// TIA Portal V18 export
// export: Created 2026-06-08T03:54:34.4007583Z, ExportSetting WithDefaults, DisplayName Totally Integrated Automation Portal, DisplayVersion V18, DisplayName TIA Portal Openness, DisplayVersion V18, DisplayName TIA Portal Version Control Interface, DisplayVersion V18, DisplayName STEP 7 Professional, DisplayVersion V18, DisplayName STEP 7 Safety, DisplayVersion V18, DisplayName WinCC Professional, DisplayVersion V18
VAR_GLOBAL   // PLC tag table "PLC_Tags"
   FT3210_Bon3 AT %ID128 : Real;   // Cảm biến lưu lượng nước dosing vào Bồn 3
   FT3210_Bon3_HMI AT %MD756 : Real;   // Giá trị mô phỏng/HMI song song cho Cảm biến lưu lượng nước dosing vào Bồn 3
   FT3210_Bon3_Use_HMI AT %M420.7 : Bool;   // Chọn chế độ mô phỏng HMI cho Cảm biến lưu lượng nước dosing vào Bồn 3
   FT3210_Bon3_Sim_Req AT %M323.0 : Bool;   // Yêu cầu mô phỏng cảm biến cho Cảm biến lưu lượng nước dosing vào Bồn 3
   FT3210_Bon3_Sim_Active AT %M323.1 : Bool;   // Mô phỏng cảm biến đang hoạt động cho Cảm biến lưu lượng nước dosing vào Bồn 3
   FT3210_Bon3_Eff AT %MD760 : Real;   // Giá trị thực tế/mô phỏng hiệu dụng cho Cảm biến lưu lượng nước dosing vào Bồn 3
   LT3213_Bon3 AT %ID132 : Real;   // Cảm biến mức liên tục Bồn 3
   LT3213_Bon3_HMI AT %MD764 : Real;   // Giá trị mô phỏng/HMI song song cho Cảm biến mức liên tục Bồn 3
   LT3213_Bon3_Use_HMI AT %M421.0 : Bool;   // Chọn chế độ mô phỏng HMI cho Cảm biến mức liên tục Bồn 3
   LT3213_Bon3_Sim_Req AT %M323.2 : Bool;   // Yêu cầu mô phỏng cảm biến cho Cảm biến mức liên tục Bồn 3
   LT3213_Bon3_Sim_Active AT %M323.3 : Bool;   // Mô phỏng cảm biến đang hoạt động cho Cảm biến mức liên tục Bồn 3
   LT3213_Bon3_Eff AT %MD768 : Real;   // Giá trị thực tế/mô phỏng hiệu dụng cho Cảm biến mức liên tục Bồn 3
   TT3214_Bon3 AT %ID136 : Real;   // Cảm biến nhiệt độ Bồn 3
   TT3214_Bon3_HMI AT %MD772 : Real;   // Giá trị mô phỏng/HMI song song cho Cảm biến nhiệt độ Bồn 3
   TT3214_Bon3_Use_HMI AT %M421.1 : Bool;   // Chọn chế độ mô phỏng HMI cho Cảm biến nhiệt độ Bồn 3
   TT3214_Bon3_Sim_Req AT %M323.4 : Bool;   // Yêu cầu mô phỏng cảm biến cho Cảm biến nhiệt độ Bồn 3
   TT3214_Bon3_Sim_Active AT %M323.5 : Bool;   // Mô phỏng cảm biến đang hoạt động cho Cảm biến nhiệt độ Bồn 3
   TT3214_Bon3_Eff AT %MD776 : Real;   // Giá trị thực tế/mô phỏng hiệu dụng cho Cảm biến nhiệt độ Bồn 3
   FT3215_Bon4 AT %ID140 : Real;   // Cảm biến lưu lượng nước dosing vào Bồn 4
   FT3215_Bon4_HMI AT %MD780 : Real;   // Giá trị mô phỏng/HMI song song cho Cảm biến lưu lượng nước dosing vào Bồn 4
   FT3215_Bon4_Use_HMI AT %M421.2 : Bool;   // Chọn chế độ mô phỏng HMI cho Cảm biến lưu lượng nước dosing vào Bồn 4
   FT3215_Bon4_Sim_Req AT %M323.6 : Bool;   // Yêu cầu mô phỏng cảm biến cho Cảm biến lưu lượng nước dosing vào Bồn 4
   FT3215_Bon4_Sim_Active AT %M323.7 : Bool;   // Mô phỏng cảm biến đang hoạt động cho Cảm biến lưu lượng nước dosing vào Bồn 4
   FT3215_Bon4_Eff AT %MD784 : Real;   // Giá trị thực tế/mô phỏng hiệu dụng cho Cảm biến lưu lượng nước dosing vào Bồn 4
   FQ3215_Bon4 AT %ID144 : Real;   // Bộ đếm lưu lượng tích lũy Bồn 4
   FQ3215_Bon4_HMI AT %MD788 : Real;   // Giá trị mô phỏng/HMI song song cho Bộ đếm lưu lượng tích lũy Bồn 4
   FQ3215_Bon4_Use_HMI AT %M421.3 : Bool;   // Chọn chế độ mô phỏng HMI cho Bộ đếm lưu lượng tích lũy Bồn 4
   FQ3215_Bon4_Sim_Req AT %M324.0 : Bool;   // Yêu cầu mô phỏng cảm biến cho Bộ đếm lưu lượng tích lũy Bồn 4
   FQ3215_Bon4_Sim_Active AT %M324.1 : Bool;   // Mô phỏng cảm biến đang hoạt động cho Bộ đếm lưu lượng tích lũy Bồn 4
   FQ3215_Bon4_Eff AT %MD792 : Real;   // Giá trị thực tế/mô phỏng hiệu dụng cho Bộ đếm lưu lượng tích lũy Bồn 4
   LS3217_Bon4_Cao AT %I0.5 : Bool;   // Cảm biến mức cao Bồn 4
   LS3217_Bon4_Cao_HMI AT %M110.5 : Bool;   // Tín hiệu mô phỏng/HMI song song cho Cảm biến mức cao Bồn 4
   LS3217_Bon4_Cao_HMI_Gated AT %M324.2 : Bool;   // Tín hiệu HMI đã qua xử lý chế độ cho Cảm biến mức cao Bồn 4
   LS3217_Bon4_Cao_Eff AT %M324.3 : Bool;   // Tín hiệu thực tế/mô phỏng hiệu dụng cho Cảm biến mức cao Bồn 4
   LT3218_Bon4 AT %ID148 : Real;   // Cảm biến mức liên tục Bồn 4
   LT3218_Bon4_HMI AT %MD796 : Real;   // Giá trị mô phỏng/HMI song song cho Cảm biến mức liên tục Bồn 4
   LT3218_Bon4_Use_HMI AT %M421.4 : Bool;   // Chọn chế độ mô phỏng HMI cho Cảm biến mức liên tục Bồn 4
   LT3218_Bon4_Sim_Req AT %M324.4 : Bool;   // Yêu cầu mô phỏng cảm biến cho Cảm biến mức liên tục Bồn 4
   LT3218_Bon4_Sim_Active AT %M324.5 : Bool;   // Mô phỏng cảm biến đang hoạt động cho Cảm biến mức liên tục Bồn 4
   LT3218_Bon4_Eff AT %MD800 : Real;   // Giá trị thực tế/mô phỏng hiệu dụng cho Cảm biến mức liên tục Bồn 4
   TT3219_Bon4 AT %ID152 : Real;   // Cảm biến nhiệt độ Bồn 4
   TT3219_Bon4_HMI AT %MD804 : Real;   // Giá trị mô phỏng/HMI song song cho Cảm biến nhiệt độ Bồn 4
   TT3219_Bon4_Use_HMI AT %M421.5 : Bool;   // Chọn chế độ mô phỏng HMI cho Cảm biến nhiệt độ Bồn 4
   TT3219_Bon4_Sim_Req AT %M324.6 : Bool;   // Yêu cầu mô phỏng cảm biến cho Cảm biến nhiệt độ Bồn 4
   TT3219_Bon4_Sim_Active AT %M324.7 : Bool;   // Mô phỏng cảm biến đang hoạt động cho Cảm biến nhiệt độ Bồn 4
   TT3219_Bon4_Eff AT %MD808 : Real;   // Giá trị thực tế/mô phỏng hiệu dụng cho Cảm biến nhiệt độ Bồn 4
   V3240_Nuoc_Bon3 AT %Q1.4 : Bool;   // Van on/off cấp nước Bồn 3
   V3240_Nuoc_Bon3_M AT %M221.4 : Bool;   // Tag gương phản hồi HMI cho Van on/off cấp nước Bồn 3
   CV3211_Nuoc_Bon3 AT %QD116 : Real;   // Van tuyến tính cấp nước Bồn 3
   CV3211_Nuoc_Bon3_M AT %MD936 : Real;   // Tag gương phản hồi HMI cho Van tuyến tính cấp nước Bồn 3
   AGTR3262_Khuay_Bon3 AT %Q1.5 : Bool;   // Động cơ khuấy Bồn 3
   AGTR3262_Khuay_Bon3_M AT %M221.5 : Bool;   // Tag gương phản hồi HMI cho Động cơ khuấy Bồn 3
   AGTR3262_Toc_Do_AO AT %QD120 : Real;   // Tín hiệu tốc độ khuấy Bồn 3
   AGTR3262_Toc_Do_AO_M AT %MD940 : Real;   // Tag gương phản hồi HMI cho Tín hiệu tốc độ khuấy Bồn 3
   V3242_Xa_Bon3 AT %Q1.6 : Bool;   // Van xả đáy Bồn 3 số 1
   V3242_Xa_Bon3_M AT %M221.6 : Bool;   // Tag gương phản hồi HMI cho Van xả đáy Bồn 3 số 1
   V3243_Xa_Bon3 AT %Q1.7 : Bool;   // Van xả đáy Bồn 3 số 2
   V3243_Xa_Bon3_M AT %M221.7 : Bool;   // Tag gương phản hồi HMI cho Van xả đáy Bồn 3 số 2
   V3244_Xa_Bon3 AT %Q2.0 : Bool;   // Van xả đáy Bồn 3 số 3
   V3244_Xa_Bon3_M AT %M222.0 : Bool;   // Tag gương phản hồi HMI cho Van xả đáy Bồn 3 số 3
   V3245_Nuoc_Bon4 AT %Q2.1 : Bool;   // Van on/off cấp nước Bồn 4
   V3245_Nuoc_Bon4_M AT %M222.1 : Bool;   // Tag gương phản hồi HMI cho Van on/off cấp nước Bồn 4
   CV3216_Hoi_Bon4 AT %QD124 : Real;   // Van tuyến tính gia nhiệt mô phỏng Bồn 4
   CV3216_Hoi_Bon4_M AT %MD944 : Real;   // Tag gương phản hồi HMI cho Van tuyến tính gia nhiệt mô phỏng Bồn 4
   AGTR3263_Khuay_Bon4 AT %Q2.2 : Bool;   // Động cơ khuấy Bồn 4
   AGTR3263_Khuay_Bon4_M AT %M222.2 : Bool;   // Tag gương phản hồi HMI cho Động cơ khuấy Bồn 4
   AGTR3263_Dao_Chieu AT %Q2.3 : Bool;   // Lệnh đảo chiều động cơ khuấy Bồn 4
   AGTR3263_Dao_Chieu_M AT %M222.3 : Bool;   // Tag gương phản hồi HMI cho Lệnh đảo chiều động cơ khuấy Bồn 4
   AGTR3263_Toc_Do_AO AT %QD128 : Real;   // Tốc độ đặt động cơ khuấy Bồn 4
   AGTR3263_Toc_Do_AO_M AT %MD948 : Real;   // Tag gương phản hồi HMI cho Tốc độ đặt động cơ khuấy Bồn 4
   V3247_Xa_Bon4 AT %Q2.4 : Bool;   // Van xả đáy Bồn 4 số 1
   V3247_Xa_Bon4_M AT %M222.4 : Bool;   // Tag gương phản hồi HMI cho Van xả đáy Bồn 4 số 1
   V3248_Xa_Bon4 AT %Q2.5 : Bool;   // Van xả đáy Bồn 4 số 2
   V3248_Xa_Bon4_M AT %M222.5 : Bool;   // Tag gương phản hồi HMI cho Van xả đáy Bồn 4 số 2
   V3249_Xa_Bon4 AT %Q2.6 : Bool;   // Van xả đáy Bồn 4 số 3
   V3249_Xa_Bon4_M AT %M222.6 : Bool;   // Tag gương phản hồi HMI cho Van xả đáy Bồn 4 số 3
   Pump3265_Chuyen_Nhanh2 AT %Q2.7 : Bool;   // Bơm chuyển dung dịch Nhánh 2 xuống bồn chứa
   Pump3265_Chuyen_Nhanh2_M AT %M222.7 : Bool;   // Tag gương phản hồi HMI cho Bơm chuyển dung dịch Nhánh 2 xuống bồn chứa
   HMI_Operator_Login AT %M422.5 : Bool;   // Đăng nhập quyền Operator
   HMI_Engineer_Login AT %M422.6 : Bool;   // Đăng nhập quyền Engineer
   HMI_Admin_Login AT %M422.7 : Bool;   // Đăng nhập quyền Admin
   HMI_Che_Do_Manual AT %M423.0 : Bool;   // Cho phép điều khiển tay từng thiết bị
   HMI_Ack_Alarm AT %M423.1 : Bool;   // Xác nhận cảnh báo
   HMI_Reset_Alarm AT %M423.2 : Bool;   // Reset alarm bằng HMI
   Gia_Lap_Mat_Ket_Noi_HMI AT %M423.3 : Bool;   // Nút giả lập mất kết nối PLC
   HMI_User_Level AT %MW520 : Int;   // Mức quyền hiện tại: 1 Operator, 2 Engineer, 3 Admin
   HMI_Cho_Phep_Sua_Thong_So AT %M327.2 : Bool;   // Cờ cho phép sửa công thức và PID
   HMI_Alarm_Status AT %MW522 : Int;   // Mã cảnh báo tổng hợp cho WinCC TextList
   HMI_AnToan_Status AT %MW524 : Int;   // Mã chẩn đoán an toàn ưu tiên
   PLC2_Auto_Enable AT %M328.1 : Bool;   // Cho phép chạy Auto Nhánh 2 Bồn 3-4
   PLC2_EStop_Latch AT %M328.2 : Bool;   // Chốt dừng khẩn HMI/SCADA Nhánh 2 Bồn 3-4
   PLC2_Loi_Tong AT %M328.3 : Bool;   // Lỗi tổng khóa Auto Nhánh 2 Bồn 3-4
   PLC2_Loi_Dry_Run AT %M328.4 : Bool;   // Lỗi chạy khô bơm Nhánh 2 Bồn 3-4
   PLC2_Loi_Dosing AT %M328.5 : Bool;   // Lỗi quá thời gian dosing Nhánh 2 Bồn 3-4
   PLC2_Loi_Truyen_Thong AT %M328.6 : Bool;   // Lỗi truyền thông mô phỏng Nhánh 2 Bồn 3-4
   PLC2_State AT %MW528 : Int;   // Mã bước chu trình Nhánh 2 Bồn 3-4
   PLC2_Step_Bon3_Dosing AT %M330.4 : Bool;   // Bồn 3 đang dosing nước
   PLC2_Step_Bon3_Tip AT %M330.5 : Bool;   // Bồn 3 đang mô phỏng tip cốt tương đậu đậm đặc
   PLC2_Step_Bon3_Khuay AT %M330.6 : Bool;   // Bồn 3 đang khuấy ban đầu
   PLC2_Step_Bon3_Xa AT %M330.7 : Bool;   // Bồn 3 đang xả sang Bồn 4
   PLC2_Step_Bon4_Dosing AT %M331.0 : Bool;   // Bồn 4 đang dosing bổ sung
   PLC2_Step_Bon4_Tip AT %M331.1 : Bool;   // Bồn 4 đang tip phụ gia
   PLC2_Step_Bon4_Khuay_Thuan AT %M331.2 : Bool;   // Bồn 4 khuấy chiều thuận
   PLC2_Step_Bon4_Khuay_Nghich AT %M331.3 : Bool;   // Bồn 4 khuấy chiều ngược
   PLC2_Step_Bon4_PID_Mo_Phong AT %M331.4 : Bool;   // Bồn 4 chạy PID mô phỏng
   PLC2_Step_Bon4_Thanh_Trung AT %M331.5 : Bool;   // Bồn 4 giữ thời gian thanh trùng
   PLC2_Xa_Bon3_Xong AT %M331.6 : Bool;   // Bồn 3 đã xả hết
   PLC2_Xa_Bon4_Xong AT %M331.7 : Bool;   // Bồn 4 đã xả hết
   PLC2_Me_Nhanh2_Hoan_Thanh AT %M332.5 : Bool;   // Cờ hoàn thành Nhánh 2 gửi sang PLC1
   PLC2_Me_Nhanh2_Hoan_Thanh_M AT %M224.6 : Bool;   // Tag gương phản hồi HMI cho cờ hoàn thành Nhánh 2 gửi sang PLC1
   Pump3265_Chuyen_Nhanh2_Cmd_Nhan AT %M333.0 : Bool;   // Nhận lệnh chạy bơm chuyển Nhánh 2 từ PLC1
   Pump3265_Chuyen_Nhanh2_Cmd_Nhan_HMI AT %M111.1 : Bool;   // Tín hiệu mô phỏng/HMI song song cho lệnh chạy bơm chuyển Nhánh 2 từ PLC1
   Nut_Khoi_Dong_Nhan AT %M333.2 : Bool;   // nút khởi động nhận từ PLC1
   Nut_Khoi_Dong_Nhan_HMI AT %M111.2 : Bool;   // Tín hiệu mô phỏng/HMI song song cho nút khởi động nhận từ PLC1
   Nut_Khoi_Dong_Nhan_HMI_Gated AT %M333.3 : Bool;   // Tín hiệu HMI đã qua xử lý chế độ cho nút khởi động nhận từ PLC1
   Nut_Khoi_Dong_Nhan_Eff AT %M333.4 : Bool;   // Tín hiệu thực tế/mô phỏng hiệu dụng cho nút khởi động nhận từ PLC1
   Nut_Dung_Nhan AT %M333.5 : Bool;   // nút dừng nhận từ PLC1
   Nut_Dung_Nhan_HMI AT %M111.3 : Bool;   // Tín hiệu mô phỏng/HMI song song cho nút dừng nhận từ PLC1
   Nut_Dung_Nhan_HMI_Gated AT %M333.6 : Bool;   // Tín hiệu HMI đã qua xử lý chế độ cho nút dừng nhận từ PLC1
   Nut_Dung_Nhan_Eff AT %M333.7 : Bool;   // Tín hiệu thực tế/mô phỏng hiệu dụng cho nút dừng nhận từ PLC1
   Nut_Reset_Nhan AT %M334.0 : Bool;   // nút reset nhận từ PLC1
   Nut_Reset_Nhan_HMI AT %M111.4 : Bool;   // Tín hiệu mô phỏng/HMI song song cho nút reset nhận từ PLC1
   Nut_Reset_Nhan_HMI_Gated AT %M334.1 : Bool;   // Tín hiệu HMI đã qua xử lý chế độ cho nút reset nhận từ PLC1
   Nut_Reset_Nhan_Eff AT %M334.2 : Bool;   // Tín hiệu thực tế/mô phỏng hiệu dụng cho nút reset nhận từ PLC1
   Nut_EStop_Nhan AT %M334.3 : Bool;   // nút dừng khẩn nhận từ PLC1
   Nut_EStop_Nhan_HMI AT %M111.5 : Bool;   // Tín hiệu mô phỏng/HMI song song cho nút dừng khẩn nhận từ PLC1
   Nut_EStop_Nhan_HMI_Gated AT %M334.4 : Bool;   // Tín hiệu HMI đã qua xử lý chế độ cho nút dừng khẩn nhận từ PLC1
   Nut_EStop_Nhan_Eff AT %M334.5 : Bool;   // Tín hiệu thực tế/mô phỏng hiệu dụng cho nút dừng khẩn nhận từ PLC1
   Clock_1Hz AT %M100.5 : Bool;   // Clock 1Hz system memory bit
   FirstScan AT %M101.0 : Bool;   // First Scan system memory bit
   PLC2_Last_CmdSeq AT %MW80 : Int;   // Last processed command sequence
   PLC2_CmdSeq_New AT %M82.0 : Bool;   // New command sequence received
   MB_TCP_Server_Error AT %M82.1 : Bool;   // Modbus TCP Server Error
   MB_TCP_Server_Status AT %MW84 : Word;   // Modbus TCP Server Status
   MB_TCP_Server_NDR AT %M82.2 : Bool;   // Modbus TCP Server New Data Received
   MB_TCP_Server_DR AT %M82.3 : Bool;   // Modbus TCP Server Data Read
   PLC1_Tip_Bon1_Xong_HMI AT %M423.4 : Bool;   // Nút mô phỏng tip Bồn 1 đã hoàn tất
   PLC1_Khuay_Bon1_Xong_HMI AT %M423.5 : Bool;   // Nút mô phỏng hết thời gian khuấy Bồn 1
   PLC1_Tip_Bon2_Xong_HMI AT %M423.6 : Bool;   // Nút mô phỏng tip Bồn 2 đã hoàn tất
   PLC1_Khuay_Thuan_Bon2_Xong_HMI AT %M423.7 : Bool;   // Nút mô phỏng hết thời gian khuấy thuận Bồn 2
   PLC1_Khuay_Nghich_Bon2_Xong_HMI AT %M424.0 : Bool;   // Nút mô phỏng hết thời gian khuấy ngược Bồn 2
   PLC1_Thanh_Trung_Bon2_Xong_HMI AT %M424.1 : Bool;   // Nút mô phỏng hết thời gian thanh trùng Bồn 2
   PLC2_Tip_Bon3_Xong_HMI AT %M424.2 : Bool;   // Nút mô phỏng tip Bồn 3 đã hoàn tất
   PLC2_Khuay_Bon3_Xong_HMI AT %M424.3 : Bool;   // Nút mô phỏng hết thời gian khuấy Bồn 3
   PLC2_Tip_Bon4_Xong_HMI AT %M424.4 : Bool;   // Nút mô phỏng tip Bồn 4 đã hoàn tất
   PLC2_Khuay_Thuan_Bon4_Xong_HMI AT %M424.5 : Bool;   // Nút mô phỏng hết thời gian khuấy thuận Bồn 4
   PLC2_Khuay_Nghich_Bon4_Xong_HMI AT %M424.6 : Bool;   // Nút mô phỏng hết thời gian khuấy ngược Bồn 4
   PLC2_Thanh_Trung_Bon4_Xong_HMI AT %M424.7 : Bool;   // Nút mô phỏng hết thời gian thanh trùng Bồn 4
   BonChua_Nhan_Dich_Xong_HMI AT %M425.0 : Bool;   // Nút mô phỏng nhận dịch vào Bồn chứa 01 xong
   BonChua_Chuyen_Bon2_Xong_HMI AT %M425.1 : Bool;   // Nút mô phỏng chuyển sang Bồn chứa 02 xong
   HMI_SP_PLC1_Nuoc_Bon1 AT %MD880 : Real;   // Lượng nước dosing Bồn 1
   HMI_SP_PLC1_Nuoc_Bon2 AT %MD884 : Real;   // Lượng nước dosing bổ sung Bồn 2
   HMI_SP_PLC1_Toc_Do_Bon1 AT %MD888 : Real;   // Tốc độ khuấy Bồn 1
   HMI_SP_PLC1_Toc_Do_Bon2_Main AT %MD892 : Real;   // Tốc độ khuấy chính Bồn 2
   HMI_SP_PLC1_Nhiet_Do_Bon2 AT %MD896 : Real;   // Setpoint nhiệt/PID Bồn 2
   HMI_SP_PLC2_Nuoc_Bon3 AT %MD900 : Real;   // Lượng nước dosing Bồn 3
   HMI_SP_PLC2_Nuoc_Bon4 AT %MD904 : Real;   // Lượng nước dosing bổ sung Bồn 4
   HMI_SP_PLC2_Toc_Do_Bon3 AT %MD908 : Real;   // Tốc độ khuấy Bồn 3
   HMI_SP_PLC2_Toc_Do_Bon4_Main AT %MD912 : Real;   // Tốc độ khuấy chính Bồn 4
   HMI_SP_PLC2_Nhiet_Do_Bon4 AT %MD916 : Real;   // Setpoint nhiệt/PID mô phỏng Bồn 4
   HMI_SP_BonChua1_Nhiet_Giai_Nhiet AT %MD920 : Real;   // Nhiệt độ giải nhiệt đích Bồn chứa 01
   HMI_SP_Loc_Ap_Suat_Max AT %MD924 : Real;   // Ngưỡng áp suất cao trước màng lọc
   HMI_SP_Time_Khuay_Bon1 AT %MD928 : Time;   // Thời gian khuấy Bồn 1
   HMI_SP_Time_Khuay_Bon3 AT %MD932 : Time;   // Thời gian khuấy Bồn 3
   HMI_SP_Time_Fwd AT %MD936 : Time;   // Thời gian khuấy chiều thuận
   HMI_SP_Time_Rev AT %MD940 : Time;   // Thời gian khuấy chiều ngược
   HMI_SP_Time_Sterilize AT %MD944 : Time;   // Thời gian giữ nhiệt thanh trùng
   PLC1_Khuay_Bon1_Xong AT %M335.3 : Bool;   // Trạng thái tự động xong khuấy Bồn 1
   PLC1_Khuay_Thuan_Bon2_Xong AT %M335.4 : Bool;   // Trạng thái tự động xong khuấy thuận Bồn 2
   PLC1_Khuay_Nghich_Bon2_Xong AT %M335.5 : Bool;   // Trạng thái tự động xong khuấy ngược Bồn 2
   PLC1_Thanh_Trung_Bon2_Xong AT %M335.6 : Bool;   // Trạng thái tự động xong thanh trùng Bồn 2
   PLC2_Khuay_Bon3_Xong AT %M335.7 : Bool;   // Trạng thái tự động xong khuấy Bồn 3
   PLC2_Khuay_Thuan_Bon4_Xong AT %M336.0 : Bool;   // Trạng thái tự động xong khuấy thuận Bồn 4
   PLC2_Khuay_Nghich_Bon4_Xong AT %M336.1 : Bool;   // Trạng thái tự động xong khuấy ngược Bồn 4
   PLC2_Thanh_Trung_Bon4_Xong AT %M336.2 : Bool;   // Trạng thái tự động xong thanh trùng Bồn 4
   PID_Bon2_Enable AT %M336.3 : Bool;   // Cho phép PID Bồn 2
   PID_Bon2_ManualEnable AT %M336.4 : Bool;   // Chế độ manual PID Bồn 2
   PID_Bon2_Error AT %M336.5 : Bool;   // Lỗi khối PID Bồn 2
   PID_Bon4_Enable AT %M336.6 : Bool;   // Cho phép PID mô phỏng Bồn 4
   PID_Bon4_ManualEnable AT %M336.7 : Bool;   // Chế độ manual PID Bồn 4
   PID_Bon4_Error AT %M337.0 : Bool;   // Lỗi khối PID Bồn 4
   PID_Bon2_ErrorBits AT %MD948 : DWord;   // Mã lỗi DWORD PID Bồn 2
   PID_Bon4_ErrorBits AT %MD952 : DWord;   // Mã lỗi DWORD PID Bồn 4
   PID_Bon2_SP AT %MD956 : Real;   // Setpoint đưa vào PID Bồn 2
   PID_Bon2_Err AT %MD960 : Real;   // Sai lệch PID Bồn 2 = SP - PV
   PID_Bon2_CV AT %MD964 : Real;   // Giá trị điều khiển PID Bồn 2
   PID_Bon2_ManualValue AT %MD968 : Real;   // Giá trị manual PID Bồn 2
   PID_Bon4_SP AT %MD972 : Real;   // Setpoint đưa vào PID mô phỏng Bồn 4
   PID_Bon4_Err AT %MD976 : Real;   // Sai lệch PID mô phỏng Bồn 4 = SP - PV
   PID_Bon4_CV AT %MD980 : Real;   // Giá trị điều khiển PID mô phỏng Bồn 4
   PID_Bon4_ManualValue AT %MD984 : Real;   // Giá trị manual PID Bồn 4
   TT3219_Bon4_Sim AT %MD988 : Real;   // Nhiệt độ mô phỏng nội bộ cho PID Bồn 4
   PID_Bon4_Tang_Nhiet_Buoc AT %MD992 : Real;   // Mức tăng nhiệt mô phỏng mỗi chu kỳ OB31
   TT3219_Bon4_Target AT %MD996 : Real;   // Nhiệt độ đích mô phỏng bồn 4
   TT3219_Bon4_Sim_Pure AT %MD1000 : Real;   // Nhiệt độ mô phỏng chưa có nhiễu bồn 4
   PID_Bon4_Temp_Val_1 AT %MD1004 : Real;   // Biến tạm mô phỏng nhiệt độ 1
   PID_Bon4_Temp_Val_2 AT %MD1008 : Real;   // Biến tạm mô phỏng nhiệt độ 2
   PID_Bon4_Sim_Counter AT %MD1012 : Real;   // Đồng hồ chu kỳ mô phỏng
   PID_Bon4_Sim_Angle AT %MD1016 : Real;   // Góc lượng giác nhiễu
   PID_Bon4_Sim_Sin AT %MD1020 : Real;   // Giá trị hình sin nhiễu
   PID_Bon4_Sim_Noise AT %MD1024 : Real;   // Giá trị nhiễu nhiệt độ
   PID_Bon4_State AT %MW536 : Int;   // Trạng thái khối PID Bồn 4
   PLC2_Stop_Active AT %M337.2 : Bool;   // Tín hiệu dừng active PLC2
   AGTR3263_Khuay_Active AT %M337.5 : Bool;   // Trạng thái khuấy Bồn 4 active
   AGTR3263_Should_Run AT %M337.6 : Bool;   // Yêu cầu chạy động cơ Bồn 4
   HMI_Use_Sim_Input_PLC2 AT %M338.0 : Bool;   // Cho phép sử dụng đầu vào mô phỏng PLC2
   Pump3265_Chuyen_Nhanh2_Cmd_Nhan_Eff AT %M338.3 : Bool;   // Lệnh chạy bơm chuyển Nhánh 2 nhận được hiệu dụng
   Pump3265_Chuyen_Nhanh2_Cmd_Nhan_HMI_Gated AT %M338.5 : Bool;   // Lệnh chạy bơm chuyển Nhánh 2 HMI gated
   PLC2_SP_Valid AT %M338.7 : Bool;   // Setpoint PLC2 hợp lệ
   PLC2_Loi_Setpoint AT %M339.2 : Bool;   // Lỗi Setpoint PLC2
   Init_Defaults_Done_PLC2 AT %M339.5 : Bool;   // Khởi tạo Setpoint mặc định PLC2 hoàn tất
   Init_Trigger_PLC2 AT %M340.0 : Bool;   // Cờ kích hoạt nạp recipe mặc định PLC2
   HMI_Load_Default_Recipe AT %M340.2 : Bool;   // Yêu cầu nạp lại Recipe mặc định từ HMI
   PLC2_Load_Default_Cmd_Nhan AT %M340.4 : Bool;   // Nhận lệnh nạp recipe mặc định từ PLC1
   PLC2_Load_Default_Cmd_Nhan_HMI AT %M111.6 : Bool;   // Tín hiệu mô phỏng/HMI cho nhận lệnh nạp recipe
   PLC2_Load_Default_Cmd_Nhan_HMI_Gated AT %M340.5 : Bool;   // Tín hiệu nhận lệnh nạp recipe HMI gated
   PLC2_Load_Default_Cmd_Nhan_Eff AT %M340.6 : Bool;   // Tín hiệu nhận lệnh nạp recipe hiệu dụng
   PLC2_Load_Default_Done AT %M340.7 : Bool;   // Báo nạp recipe mặc định xong gửi sang PLC1
   PLC2_Load_Default_Done_M AT %M225.1 : Bool;   // Tag gương phản hồi HMI cho báo nạp recipe xong PLC2
   HMI_Sim_Mode AT %M341.3 : Bool;   // Cho phép toàn bộ tín hiệu mô phỏng HMI tác động vào input hiệu dụng
   HMI_Run_Enable AT %M341.4 : Bool;   // Cho phép vận hành từ HMI ở chế độ thật
   System_Mode_Real AT %M341.5 : Bool;   // Hệ thống đang hoạt động ở chế độ thực tế
   System_Mode_Sim AT %M341.6 : Bool;   // Hệ thống đang hoạt động ở chế độ mô phỏng
   HMI_Sim_Active_Warning AT %M341.7 : Bool;   // Cảnh báo chế độ mô phỏng HMI đang hoạt động
END_VAR
